(* PLC project v0.6.04_CycleSemiAuto.project, CODESYS CODESYS V3.5 SP19 Patch 1 *)
(* stored: creationDateTime 2026-07-26T19:54:07.376406, modificationDateTime 2026-07-26T19:54:07.376406 *)

(* ═══════════════════════════════════════════════════════════════ 🔧 ST_BypassSync — Bypass de la surveillance synchronisation M1/M2 🔒 Doctrine : actionnable UNIQUEMENT en MAINT_N2, RETAIN, jamais masque les autres défauts du même bloc (voir REGISTRE_ACTIONS_Bypass_v1.0 (archive)). ═══════════════════════════════════════════════════════════════ *)
TYPE ST_BypassSync : STRUCT
  Global : BOOL := FALSE;  (* 🌐 Bypass GLOBAL synchro : ignore toute erreur de synchronisation *)
  Initialized : BOOL := FALSE;  (* 🚦 flag restauration boot *)
END_STRUCT;
END_TYPE
